// TIA Portal project "TestCase4_S1500_Met_Fouten" (V18)

(* hardware
DEVICE "S7-1500/ET200MP station_1"  S7-1500 station
   slot 0: "Rail_0"  Rack  6ES7 590-1***0-0AA0
   slot 1: "PLC_1"  CPU 1511C-1 PN  6ES7 511-1CK00-0AB0  V2.9
      slot 3: "CPU display_1"  6ES7591-1AA00-0AA0
      slot 32768: "PROFINET interface_1"  X1
         slot 32769: "Port_1"  X1 P1
         slot 32770: "Port_2"  X1 P2
      slot 34817: "Virtual CP interface port_1"  Virtual CP interface port  Virtual CP interface port
*)

// ===== PLC "PLC_1"  CPU 1511C-1 PN =====

VAR_GLOBAL   // PLC tag table "Default tag table"
   "Tag_3" AT %M100.1 : Bool;
   "Tag_4" AT %M100.0 : Bool;
   "Tag_1" AT %M101.0 : Bool;
   "Tag_5" AT %M102.0 : Bool;
   "Tag_6" AT %M101.1 : Bool;
   "Tag_7" AT %M103.0 : Bool;
   "sensor1" AT %I0.0 : Bool;
   "sensor2" AT %I0.1 : Bool;
   "sensor3" AT %I0.2 : Bool;
   "lampA" AT %Q0.0 : Bool;
   "lampB" AT %Q0.1 : Bool;
   "Tag_8" AT %M100.2 : Bool;
   "Tag_9" AT %M103.1 : Bool;
END_VAR

DATA_BLOCK "Data_block_1"   // DB1
{ S7_Optimized_Access := 'FALSE' }
VERSION : 0.1
   VAR
      sensor1 : Bool;
      sensor2 : Bool;
      sensor3 : Bool;
   END_VAR
BEGIN
END_DATA_BLOCK

DATA_BLOCK "Data_block_2"   // DB2
{ S7_Optimized_Access := 'FALSE' }
VERSION : 0.1
   VAR
      lampA : Bool;
      lampB : Bool;
   END_VAR
BEGIN
END_DATA_BLOCK

FUNCTION "State0" : Void   // FC1, FBD
{ S7_Optimized_Access := 'TRUE' }
VERSION : 0.1
BEGIN

REGION Network 1
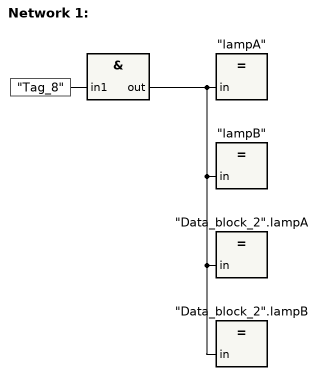
   "lampA" := "Tag_8";
   "lampB" := "Tag_8";
   "Data_block_2".lampA := "Tag_8";
   "Data_block_2".lampB := "Tag_8";
END_REGION
END_FUNCTION

FUNCTION "State1" : Void   // FC2, FBD
{ S7_Optimized_Access := 'TRUE' }
VERSION : 0.1
BEGIN

REGION Network 1
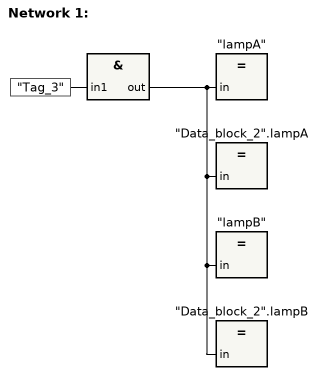
   "lampA" := "Tag_3";
   "Data_block_2".lampA := "Tag_3";
   "lampB" := "Tag_3";
   "Data_block_2".lampB := "Tag_3";
END_REGION
END_FUNCTION

FUNCTION "State2" : Void   // FC3, FBD
{ S7_Optimized_Access := 'TRUE' }
VERSION : 0.1
BEGIN

REGION Network 1
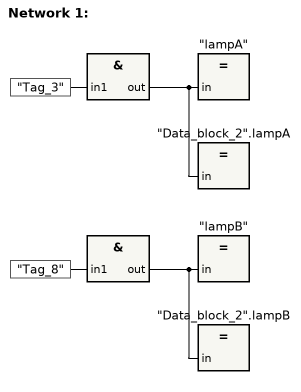
   "lampA" := "Tag_3";
   "Data_block_2".lampA := "Tag_3";
   "lampB" := "Tag_8";
   "Data_block_2".lampB := "Tag_8";
END_REGION
END_FUNCTION

ORGANIZATION_BLOCK "Main"   // OB1, FBD, ProgramCycle
TITLE = "Main Program Sweep (Cycle)"
{ S7_Optimized_Access := 'FALSE' }
VERSION : 0.1
   VAR_TEMP
      EV_CLASS : Byte;   // Bits 0-3 = 1:Coming event, Bits 4-7 = 1:Event class 1
      SCAN_1 : Byte;   // 1:Initial call of the OB, 3: Call 2-n of the OB
      PRIORITY : Byte;   // Priority of OB Execution
      OB_NUMBR : Byte;   // OB number
      RESERVED_1 : Byte;   // Reserved for system
      RESERVED_2 : Byte;   // Reserved for system
      PREV_CYCLE : Int;   // Previous program cycle time (milliseconds)
      MIN_CYCLE : Int;   // Minimum program cycle time (milliseconds)
      MAX_CYCLE : Int;   // Maximum program cycle time (milliseconds)
      DATE_TIME : Date_And_Time;   // Date and time OB started
   END_VAR
BEGIN

REGION Network 1
   // Initialize Merkers (M100.0 = 1 cycle true, M100.1 always 1 and M100.2 always 0).
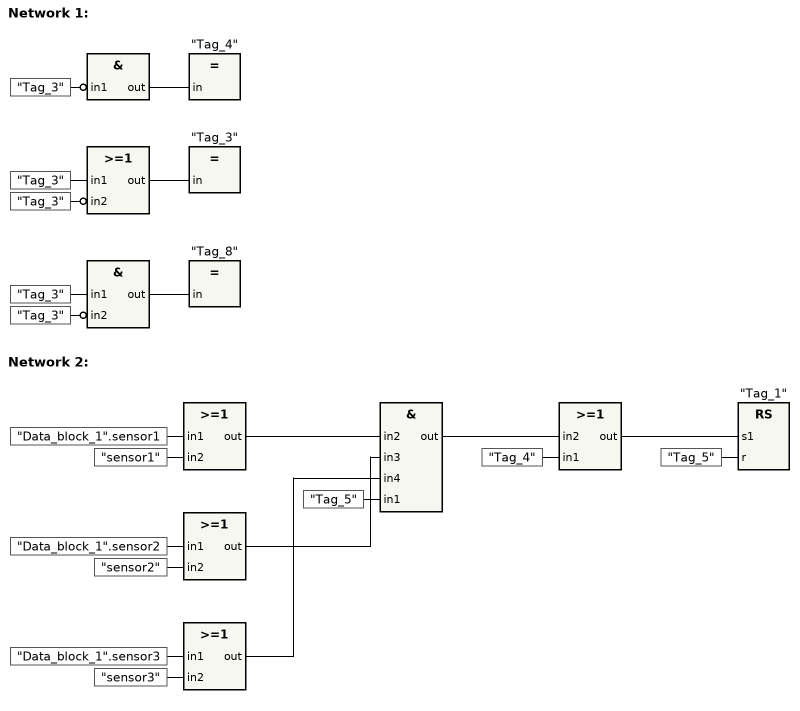
   "Tag_4" := NOT "Tag_3";
   "Tag_3" := "Tag_3" OR NOT "Tag_3";
   "Tag_8" := "Tag_3" AND NOT "Tag_3";
END_REGION

REGION Network 2
   // State 0
   IF "Tag_5" THEN
       "Tag_1" := FALSE;   // RS flip-flop
   END_IF;
   IF (("Data_block_1".sensor1 OR "sensor1") AND ("Data_block_1".sensor2 OR "sensor2") AND ("Data_block_1".sensor3 OR "sensor3") AND "Tag_5") OR "Tag_4" THEN
       "Tag_1" := TRUE;
   END_IF;
END_REGION

REGION Network 3
   // State 1
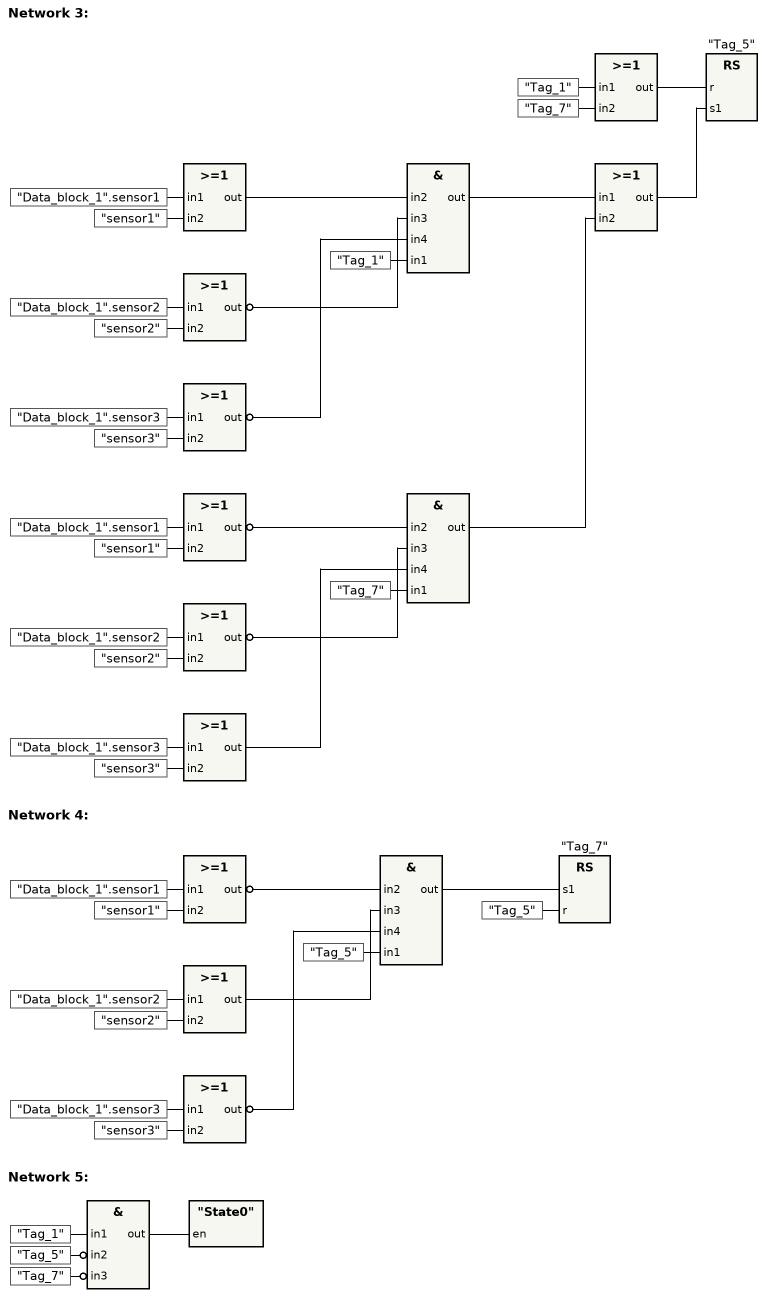
   IF "Tag_1" OR "Tag_7" THEN
       "Tag_5" := FALSE;   // RS flip-flop
   END_IF;
   IF (("Data_block_1".sensor1 OR "sensor1") AND NOT ("Data_block_1".sensor2 OR "sensor2") AND NOT ("Data_block_1".sensor3 OR "sensor3") AND "Tag_1") OR (NOT ("Data_block_1".sensor1 OR "sensor1") AND NOT ("Data_block_1".sensor2 OR "sensor2") AND ("Data_block_1".sensor3 OR "sensor3") AND "Tag_7") THEN
       "Tag_5" := TRUE;
   END_IF;
END_REGION

REGION Network 4
   // State 2
   IF "Tag_5" THEN
       "Tag_7" := FALSE;   // RS flip-flop
   END_IF;
   IF NOT ("Data_block_1".sensor1 OR "sensor1") AND ("Data_block_1".sensor2 OR "sensor2") AND NOT ("Data_block_1".sensor3 OR "sensor3") AND "Tag_5" THEN
       "Tag_7" := TRUE;
   END_IF;
END_REGION

REGION Network 5
   // Activate the outputs
   IF "Tag_1" AND NOT "Tag_5" AND NOT "Tag_7" THEN "State0"(); END_IF;
END_REGION

REGION Network 6
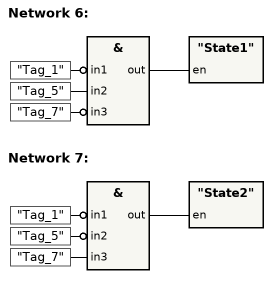
   IF NOT "Tag_1" AND "Tag_5" AND NOT "Tag_7" THEN "State1"(); END_IF;
END_REGION

REGION Network 7
   IF NOT "Tag_1" AND NOT "Tag_5" AND "Tag_7" THEN "State2"(); END_IF;
END_REGION
END_ORGANIZATION_BLOCK